TYPE ST_WZ_Zustand :
STRUCT
	Volumen				: REAL;
	Freigabe				: BOOL;
	Temperatur_Vorlauf		: REAL;
	Temperatur_Ruecklauf	: REAL;
	Volumenstrom			: REAL;
	Energie					: REAL;
	Leistung				: REAL;
	Temperatur_Diff			: REAL;
END_STRUCT
END_TYPE

(* stored: Version 1.1.0.1, ProductVersion 3.1.4024.9
   DUT ST_WZ_Zustand: Id {dda7cbe4-cb43-4383-887d-51f3a953a734} *)
